// TIA Portal V17 export
// export: Created 2022-03-12T16:05:31.0251124Z, ExportSetting WithDefaults, DisplayName Totally Integrated Automation Portal, DisplayVersion V17, DisplayName TIA Portal Openness, DisplayVersion V17, DisplayName TIA Portal Version Control Interface, DisplayVersion V17, DisplayName STEP 7 Professional, DisplayVersion V17, DisplayName STEP 7 Safety, DisplayVersion V17, DisplayName WinCC Advanced / Unified PC, DisplayVersion V17
DATA_BLOCK "PackML"   // DB31613
TITLE = CPG_PackML
{ S7_Optimized_Access := 'TRUE' }
AUTHOR : tech.team.motioncontrol@siemens.com
FAMILY : CPG
VERSION : 1.0
// Support: tech.team.motioncontrol@siemens.com
// Fax: +49 (0) 9131/98-1297
// stored: AutoNumber true, DBAccessibleFromOPCUA true, DBAccessibleFromWebserver true, IsOnlyStoredInLoadMemory false, IsRetainMemResEnabled false, IsWriteProtectedInAS false, MemoryReserve 0
   VAR
      projectVersion { ExternalWritable := 'False'} : String[10] := 'V1.0.0';   // Project specific version
      Cmd : Struct   // PackML boolean COMMAND to PackML ModeManager & State Model
         Mode : Struct   // Boolean command to change the MODE
            Production : Bool;   // Request to goto mode - PRODUCTION (mode #1)
            Maintenance : Bool;   // Request to goto mode - MAINTENANCE (mode #2)
            Manual : Bool;   // Request to goto mode - MANUAL (mode #3)
            UserMode01 : Bool;   // Request to goto mode - USER MODE 01 (mode #4)
            UserMode02 : Bool;   // Request to goto mode - USER MODE 02 (mode #5)
            UserMode03 : Bool;   // Request to goto mode - USER MODE 03 (mode #6)
            UserMode04 : Bool;   // Request to goto mode - USER MODE 04 (mode #7)
            UserMode05 : Bool;   // Request to goto mode - USER MODE 05 (mode #8)
            UserMode06 : Bool;   // Request to goto mode - USER MODE 06 (mode #9)
            UserMode07 : Bool;   // Request to goto mode - USER MODE 07 (mode #10)
            UserMode08 : Bool;   // Request to goto mode - USER MODE 08 (mode #11)
         END_STRUCT;
      END_STRUCT;
      Sts { ExternalWritable := 'False'} : Struct   // Status for current mode and state as boolean
         Mode { ExternalWritable := 'False'} : Struct   // Status of the current MODE
            Production { ExternalWritable := 'False'} : Bool;   // Current mode - PRODUCTION (mode #1)
            Maintenance { ExternalWritable := 'False'} : Bool;   // Current mode - MAINTENANCE (mode #2)
            Manual { ExternalWritable := 'False'} : Bool;   // Current mode - MANUAL (mode #3)
            UserMode01 { ExternalWritable := 'False'} : Bool;   // Current mode - USER MODE 01 (mode #4)
            UserMode02 { ExternalWritable := 'False'} : Bool;   // Current mode - USER MODE 02 (mode #5)
            UserMode03 { ExternalWritable := 'False'} : Bool;   // Current mode - USER MODE 03 (mode #6)
            UserMode04 { ExternalWritable := 'False'} : Bool;   // Current mode - USER MODE 04 (mode #7)
            UserMode05 { ExternalWritable := 'False'} : Bool;   // Current mode - USER MODE 05 (mode #8)
            UserMode06 { ExternalWritable := 'False'} : Bool;   // Current mode - USER MODE 06 (mode #9)
            UserMode07 { ExternalWritable := 'False'} : Bool;   // Current mode - USER MODE 07 (mode #10)
            UserMode08 { ExternalWritable := 'False'} : Bool;   // Current mode - USER MODE 08 (mode #11)
         END_STRUCT;
         State { ExternalWritable := 'False'} : Struct   // Status of the current STATE
            Clearing { ExternalWritable := 'False'} : Bool;   // Current state is - Clearing
            Stopped { ExternalWritable := 'False'} : Bool;   // Current state is - Stopped
            Starting { ExternalWritable := 'False'} : Bool;   // Current state is - Starting
            Idle { ExternalWritable := 'False'} : Bool;   // Current state is - Idle
            Suspended { ExternalWritable := 'False'} : Bool;   // Current state is - Suspended
            Execute { ExternalWritable := 'False'} : Bool;   // Current state is - Executing
            Stopping { ExternalWritable := 'False'} : Bool;   // Current state is - Stopping
            Aborting { ExternalWritable := 'False'} : Bool;   // Current state is - Aborting
            Aborted { ExternalWritable := 'False'} : Bool;   // Current state is - Aborted
            Holding { ExternalWritable := 'False'} : Bool;   // Current state is - Holding
            Held { ExternalWritable := 'False'} : Bool;   // Current state is - Held
            Unholding { ExternalWritable := 'False'} : Bool;   // Current state is - Unholding
            Suspending { ExternalWritable := 'False'} : Bool;   // Current state is - Suspending
            Unsuspending { ExternalWritable := 'False'} : Bool;   // Current state is - Unsuspending
            Resetting { ExternalWritable := 'False'} : Bool;   // Current state is - Resetting
            Completing { ExternalWritable := 'False'} : Bool;   // Current state is - Completing
            Complete { ExternalWritable := 'False'} : Bool;   // Current state is - Complete
         END_STRUCT;
      END_STRUCT;
      Cmd_Reset : Bool;   // Request for command - RESET
      Cmd_Start : Bool;   // Request for command - START
      Cmd_Stop : Bool;   // Request for command - STOP
      Cmd_Hold : Bool;   // Request for command - HOLD
      Cmd_UnHold : Bool;   // Request for command - UNHOLD
      Cmd_Suspend : Bool;   // Request for command - SUSPEND
      Cmd_UnSuspend : Bool;   // Request for command - UNSUSPEND
      Cmd_Abort : Bool;   // Request for command - ABORT
      Cmd_Clear : Bool;   // Request for command - CLEAR
      Cmd_Complete : Bool;   // Request for command - COMPLETE
      remoteCommandEnable : Bool;   // If 0 = local mode for PackML commands, if 1=remote command for PackML
      OEE { ExternalWritable := 'False'} : Struct   // Real-Time OEE values
         realTime { ExternalWritable := 'False'} : Real;   // Real-Time value (0-100%)
         availability { ExternalWritable := 'False'} : Real;   // Availability value (0-100%)
         performance { ExternalWritable := 'False'} : Real;   // Performance value (0-100%)
         quality { ExternalWritable := 'False'} : Real;   // Quality value (0-100%)
      END_STRUCT;
      PackMLDiag { ExternalWritable := 'False'; S7_SetPoint := 'True'} : "typeLPMLV30_Diagnostics";   // PackML Diagnostic Data
   END_VAR
BEGIN
END_DATA_BLOCK
